TYPE "TAx_Speed_Alarms"
VERSION : 0.1
// Block: TAx_Speed_Alarms
   STRUCT
      TOAxis : Bool;
      MCFunction : Bool;
      Drive : Bool;
   END_STRUCT;

END_TYPE
